# EPICS autosave request: iocBoot/sioc-esb-hppm1/hp8xxxa.req
file "../commonSettings.req", P=$(P)
